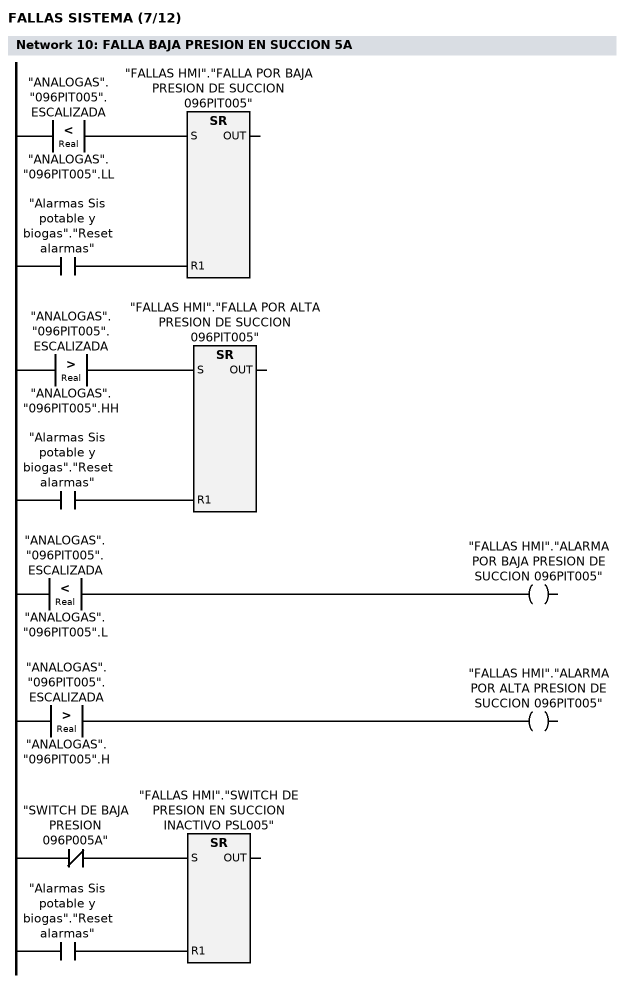
   RUNG wire#powerrail
      { S7_Templates := "SrcType := Real" } LT_Contact(in1 := "ANALOGAS"."096PIT005".ESCALIZADA, in2 := "ANALOGAS"."096PIT005".LL)
      S_SR(operand := "FALLAS HMI"."FALLA POR BAJA PRESION DE SUCCION 096PIT005", r1 := wire#w1)
   END_RUNG
   RUNG wire#powerrail
      Contact( "Alarmas Sis potable y biogas"."Reset alarmas" )
   END_RUNG wire#w1
   RUNG wire#powerrail
      { S7_Templates := "SrcType := Real" } GT_Contact(in1 := "ANALOGAS"."096PIT005".ESCALIZADA, in2 := "ANALOGAS"."096PIT005".HH)
      S_SR(operand := "FALLAS HMI"."FALLA POR ALTA PRESION DE SUCCION 096PIT005", r1 := wire#w2)
   END_RUNG
   RUNG wire#powerrail
      Contact( "Alarmas Sis potable y biogas"."Reset alarmas" )
   END_RUNG wire#w2
   RUNG wire#powerrail
      { S7_Templates := "SrcType := Real" } LT_Contact(in1 := "ANALOGAS"."096PIT005".ESCALIZADA, in2 := "ANALOGAS"."096PIT005".L)
      Coil( "FALLAS HMI"."ALARMA POR BAJA PRESION DE SUCCION 096PIT005" )
   END_RUNG
   RUNG wire#powerrail
      { S7_Templates := "SrcType := Real" } GT_Contact(in1 := "ANALOGAS"."096PIT005".ESCALIZADA, in2 := "ANALOGAS"."096PIT005".H)
      Coil( "FALLAS HMI"."ALARMA POR ALTA PRESION DE SUCCION 096PIT005" )
   END_RUNG
   RUNG wire#powerrail
      I_Contact( "SWITCH DE BAJA PRESION 096P005A" )
      S_SR(operand := "FALLAS HMI"."SWITCH DE PRESION EN SUCCION INACTIVO PSL005", r1 := wire#w3)
   END_RUNG
   RUNG wire#powerrail
      Contact( "Alarmas Sis potable y biogas"."Reset alarmas" )
   END_RUNG wire#w3
   // the same network as SCL:
   IF "ANALOGAS"."096PIT005".ESCALIZADA < "ANALOGAS"."096PIT005".LL THEN
       "FALLAS HMI"."FALLA POR BAJA PRESION DE SUCCION 096PIT005" := TRUE;   // SR flip-flop
   END_IF;
   IF "Alarmas Sis potable y biogas"."Reset alarmas" THEN
       "FALLAS HMI"."FALLA POR BAJA PRESION DE SUCCION 096PIT005" := FALSE;
   END_IF;
   IF "ANALOGAS"."096PIT005".ESCALIZADA > "ANALOGAS"."096PIT005".HH THEN
       "FALLAS HMI"."FALLA POR ALTA PRESION DE SUCCION 096PIT005" := TRUE;   // SR flip-flop
   END_IF;
   IF "Alarmas Sis potable y biogas"."Reset alarmas" THEN
       "FALLAS HMI"."FALLA POR ALTA PRESION DE SUCCION 096PIT005" := FALSE;
   END_IF;
   "FALLAS HMI"."ALARMA POR BAJA PRESION DE SUCCION 096PIT005" := "ANALOGAS"."096PIT005".ESCALIZADA < "ANALOGAS"."096PIT005".L;
   "FALLAS HMI"."ALARMA POR ALTA PRESION DE SUCCION 096PIT005" := "ANALOGAS"."096PIT005".ESCALIZADA > "ANALOGAS"."096PIT005".H;
   IF NOT "SWITCH DE BAJA PRESION 096P005A" THEN
       "FALLAS HMI"."SWITCH DE PRESION EN SUCCION INACTIVO PSL005" := TRUE;   // SR flip-flop
   END_IF;
   IF "Alarmas Sis potable y biogas"."Reset alarmas" THEN
       "FALLAS HMI"."SWITCH DE PRESION EN SUCCION INACTIVO PSL005" := FALSE;
   END_IF;
END_REGION

REGION Network 11: FALLA BAJA PRESION EN SUCCION 5B
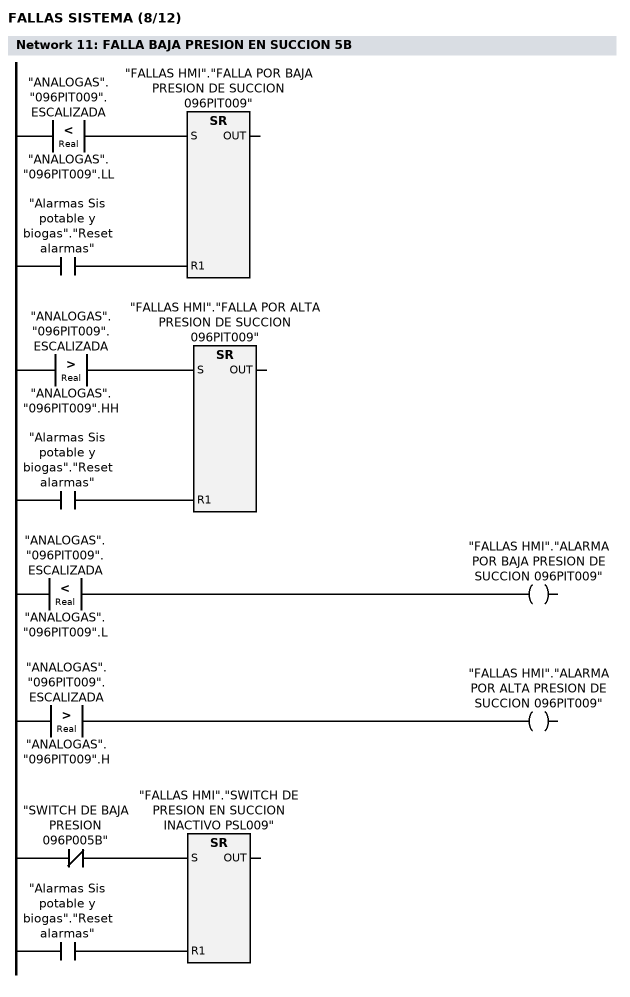
   RUNG wire#powerrail
      { S7_Templates := "SrcType := Real" } LT_Contact(in1 := "ANALOGAS"."096PIT009".ESCALIZADA, in2 := "ANALOGAS"."096PIT009".LL)
      S_SR(operand := "FALLAS HMI"."FALLA POR BAJA PRESION DE SUCCION 096PIT009", r1 := wire#w1)
   END_RUNG
   RUNG wire#powerrail
      Contact( "Alarmas Sis potable y biogas"."Reset alarmas" )
   END_RUNG wire#w1
   RUNG wire#powerrail
      { S7_Templates := "SrcType := Real" } GT_Contact(in1 := "ANALOGAS"."096PIT009".ESCALIZADA, in2 := "ANALOGAS"."096PIT009".HH)
      S_SR(operand := "FALLAS HMI"."FALLA POR ALTA PRESION DE SUCCION 096PIT009", r1 := wire#w2)
   END_RUNG
   RUNG wire#powerrail
      Contact( "Alarmas Sis potable y biogas"."Reset alarmas" )
   END_RUNG wire#w2
   RUNG wire#powerrail
      { S7_Templates := "SrcType := Real" } LT_Contact(in1 := "ANALOGAS"."096PIT009".ESCALIZADA, in2 := "ANALOGAS"."096PIT009".L)
      Coil( "FALLAS HMI"."ALARMA POR BAJA PRESION DE SUCCION 096PIT009" )
   END_RUNG
   RUNG wire#powerrail
      { S7_Templates := "SrcType := Real" } GT_Contact(in1 := "ANALOGAS"."096PIT009".ESCALIZADA, in2 := "ANALOGAS"."096PIT009".H)
      Coil( "FALLAS HMI"."ALARMA POR ALTA PRESION DE SUCCION 096PIT009" )
   END_RUNG
   RUNG wire#powerrail
      I_Contact( "SWITCH DE BAJA PRESION 096P005B" )
      S_SR(operand := "FALLAS HMI"."SWITCH DE PRESION EN SUCCION INACTIVO PSL009", r1 := wire#w3)
   END_RUNG
   RUNG wire#powerrail
      Contact( "Alarmas Sis potable y biogas"."Reset alarmas" )
   END_RUNG wire#w3
   // the same network as SCL:
   IF "ANALOGAS"."096PIT009".ESCALIZADA < "ANALOGAS"."096PIT009".LL THEN
       "FALLAS HMI"."FALLA POR BAJA PRESION DE SUCCION 096PIT009" := TRUE;   // SR flip-flop
   END_IF;
   IF "Alarmas Sis potable y biogas"."Reset alarmas" THEN
       "FALLAS HMI"."FALLA POR BAJA PRESION DE SUCCION 096PIT009" := FALSE;
   END_IF;
   IF "ANALOGAS"."096PIT009".ESCALIZADA > "ANALOGAS"."096PIT009".HH THEN
       "FALLAS HMI"."FALLA POR ALTA PRESION DE SUCCION 096PIT009" := TRUE;   // SR flip-flop
   END_IF;
   IF "Alarmas Sis potable y biogas"."Reset alarmas" THEN
       "FALLAS HMI"."FALLA POR ALTA PRESION DE SUCCION 096PIT009" := FALSE;
   END_IF;
   "FALLAS HMI"."ALARMA POR BAJA PRESION DE SUCCION 096PIT009" := "ANALOGAS"."096PIT009".ESCALIZADA < "ANALOGAS"."096PIT009".L;
   "FALLAS HMI"."ALARMA POR ALTA PRESION DE SUCCION 096PIT009" := "ANALOGAS"."096PIT009".ESCALIZADA > "ANALOGAS"."096PIT009".H;
   IF NOT "SWITCH DE BAJA PRESION 096P005B" THEN
       "FALLAS HMI"."SWITCH DE PRESION EN SUCCION INACTIVO PSL009" := TRUE;   // SR flip-flop
   END_IF;
   IF "Alarmas Sis potable y biogas"."Reset alarmas" THEN
       "FALLAS HMI"."SWITCH DE PRESION EN SUCCION INACTIVO PSL009" := FALSE;
   END_IF;
END_REGION

REGION Network 12: FALLA BAJA PRESION EN DESCARGA POTABLE
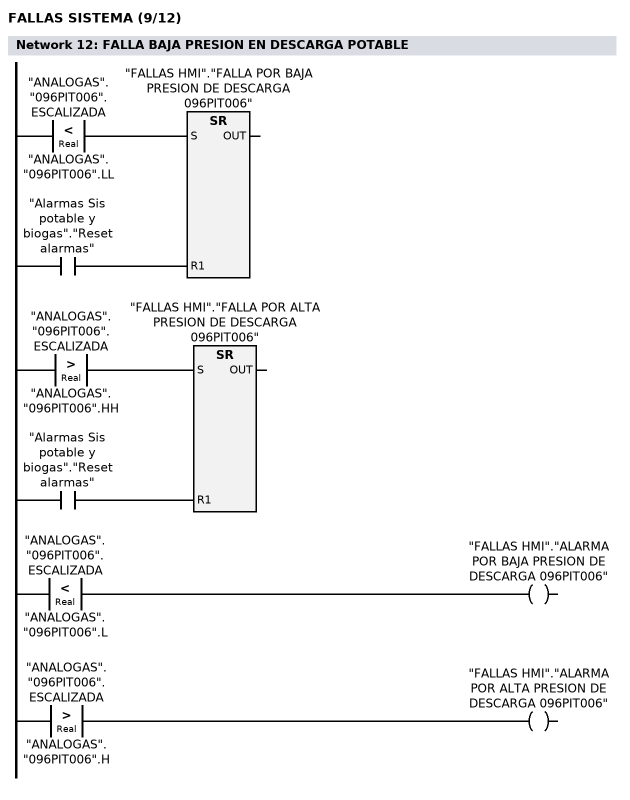
   RUNG wire#powerrail
      { S7_Templates := "SrcType := Real" } LT_Contact(in1 := "ANALOGAS"."096PIT006".ESCALIZADA, in2 := "ANALOGAS"."096PIT006".LL)
      S_SR(operand := "FALLAS HMI"."FALLA POR BAJA PRESION DE DESCARGA 096PIT006", r1 := wire#w1)
   END_RUNG
   RUNG wire#powerrail
      Contact( "Alarmas Sis potable y biogas"."Reset alarmas" )
   END_RUNG wire#w1
   RUNG wire#powerrail
      { S7_Templates := "SrcType := Real" } GT_Contact(in1 := "ANALOGAS"."096PIT006".ESCALIZADA, in2 := "ANALOGAS"."096PIT006".HH)
      S_SR(operand := "FALLAS HMI"."FALLA POR ALTA PRESION DE DESCARGA 096PIT006", r1 := wire#w2)
   END_RUNG
   RUNG wire#powerrail
      Contact( "Alarmas Sis potable y biogas"."Reset alarmas" )
   END_RUNG wire#w2
   RUNG wire#powerrail
      { S7_Templates := "SrcType := Real" } LT_Contact(in1 := "ANALOGAS"."096PIT006".ESCALIZADA, in2 := "ANALOGAS"."096PIT006".L)
      Coil( "FALLAS HMI"."ALARMA POR BAJA PRESION DE DESCARGA 096PIT006" )
   END_RUNG
   RUNG wire#powerrail
      { S7_Templates := "SrcType := Real" } GT_Contact(in1 := "ANALOGAS"."096PIT006".ESCALIZADA, in2 := "ANALOGAS"."096PIT006".H)
      Coil( "FALLAS HMI"."ALARMA POR ALTA PRESION DE DESCARGA 096PIT006" )
   END_RUNG
   // the same network as SCL:
   IF "ANALOGAS"."096PIT006".ESCALIZADA < "ANALOGAS"."096PIT006".LL THEN
       "FALLAS HMI"."FALLA POR BAJA PRESION DE DESCARGA 096PIT006" := TRUE;   // SR flip-flop
   END_IF;
   IF "Alarmas Sis potable y biogas"."Reset alarmas" THEN
       "FALLAS HMI"."FALLA POR BAJA PRESION DE DESCARGA 096PIT006" := FALSE;
   END_IF;
   IF "ANALOGAS"."096PIT006".ESCALIZADA > "ANALOGAS"."096PIT006".HH THEN
       "FALLAS HMI"."FALLA POR ALTA PRESION DE DESCARGA 096PIT006" := TRUE;   // SR flip-flop
   END_IF;
   IF "Alarmas Sis potable y biogas"."Reset alarmas" THEN
       "FALLAS HMI"."FALLA POR ALTA PRESION DE DESCARGA 096PIT006" := FALSE;
   END_IF;
   "FALLAS HMI"."ALARMA POR BAJA PRESION DE DESCARGA 096PIT006" := "ANALOGAS"."096PIT006".ESCALIZADA < "ANALOGAS"."096PIT006".L;
   "FALLAS HMI"."ALARMA POR ALTA PRESION DE DESCARGA 096PIT006" := "ANALOGAS"."096PIT006".ESCALIZADA > "ANALOGAS"."096PIT006".H;
END_REGION

REGION Network 13: FALLA BAJA PRESION EN DESCARGA 5A
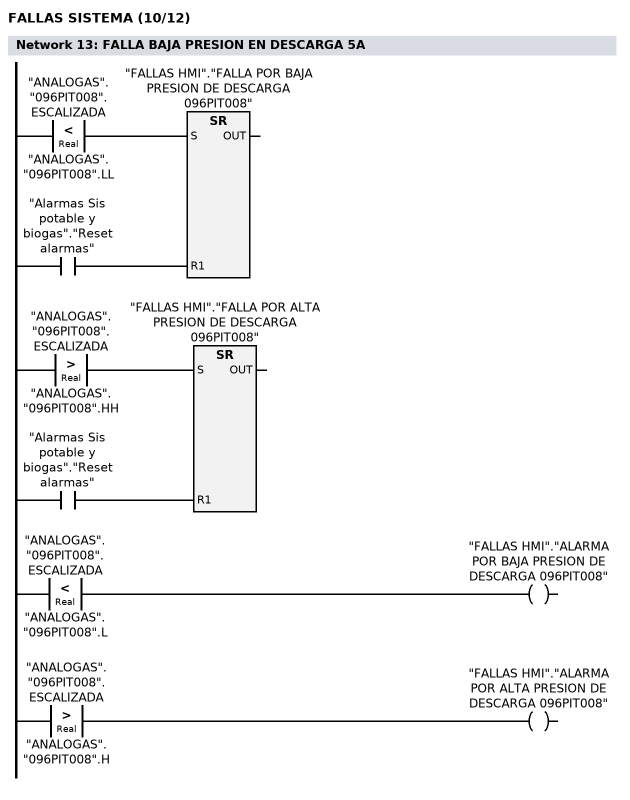
   RUNG wire#powerrail
      { S7_Templates := "SrcType := Real" } LT_Contact(in1 := "ANALOGAS"."096PIT008".ESCALIZADA, in2 := "ANALOGAS"."096PIT008".LL)
      S_SR(operand := "FALLAS HMI"."FALLA POR BAJA PRESION DE DESCARGA 096PIT008", r1 := wire#w1)
   END_RUNG
   RUNG wire#powerrail
      Contact( "Alarmas Sis potable y biogas"."Reset alarmas" )
   END_RUNG wire#w1
   RUNG wire#powerrail
      { S7_Templates := "SrcType := Real" } GT_Contact(in1 := "ANALOGAS"."096PIT008".ESCALIZADA, in2 := "ANALOGAS"."096PIT008".HH)
      S_SR(operand := "FALLAS HMI"."FALLA POR ALTA PRESION DE DESCARGA 096PIT008", r1 := wire#w2)
   END_RUNG
   RUNG wire#powerrail
      Contact( "Alarmas Sis potable y biogas"."Reset alarmas" )
   END_RUNG wire#w2
   RUNG wire#powerrail
      { S7_Templates := "SrcType := Real" } LT_Contact(in1 := "ANALOGAS"."096PIT008".ESCALIZADA, in2 := "ANALOGAS"."096PIT008".L)
      Coil( "FALLAS HMI"."ALARMA POR BAJA PRESION DE DESCARGA 096PIT008" )
   END_RUNG
   RUNG wire#powerrail
      { S7_Templates := "SrcType := Real" } GT_Contact(in1 := "ANALOGAS"."096PIT008".ESCALIZADA, in2 := "ANALOGAS"."096PIT008".H)
      Coil( "FALLAS HMI"."ALARMA POR ALTA PRESION DE DESCARGA 096PIT008" )
   END_RUNG
   // the same network as SCL:
   IF "ANALOGAS"."096PIT008".ESCALIZADA < "ANALOGAS"."096PIT008".LL THEN
       "FALLAS HMI"."FALLA POR BAJA PRESION DE DESCARGA 096PIT008" := TRUE;   // SR flip-flop
   END_IF;
   IF "Alarmas Sis potable y biogas"."Reset alarmas" THEN
       "FALLAS HMI"."FALLA POR BAJA PRESION DE DESCARGA 096PIT008" := FALSE;
   END_IF;
   IF "ANALOGAS"."096PIT008".ESCALIZADA > "ANALOGAS"."096PIT008".HH THEN
       "FALLAS HMI"."FALLA POR ALTA PRESION DE DESCARGA 096PIT008" := TRUE;   // SR flip-flop
   END_IF;
   IF "Alarmas Sis potable y biogas"."Reset alarmas" THEN
       "FALLAS HMI"."FALLA POR ALTA PRESION DE DESCARGA 096PIT008" := FALSE;
   END_IF;
   "FALLAS HMI"."ALARMA POR BAJA PRESION DE DESCARGA 096PIT008" := "ANALOGAS"."096PIT008".ESCALIZADA < "ANALOGAS"."096PIT008".L;
   "FALLAS HMI"."ALARMA POR ALTA PRESION DE DESCARGA 096PIT008" := "ANALOGAS"."096PIT008".ESCALIZADA > "ANALOGAS"."096PIT008".H;
END_REGION

REGION Network 14: FALLA BAJA PRESION EN DESCARGA 5B
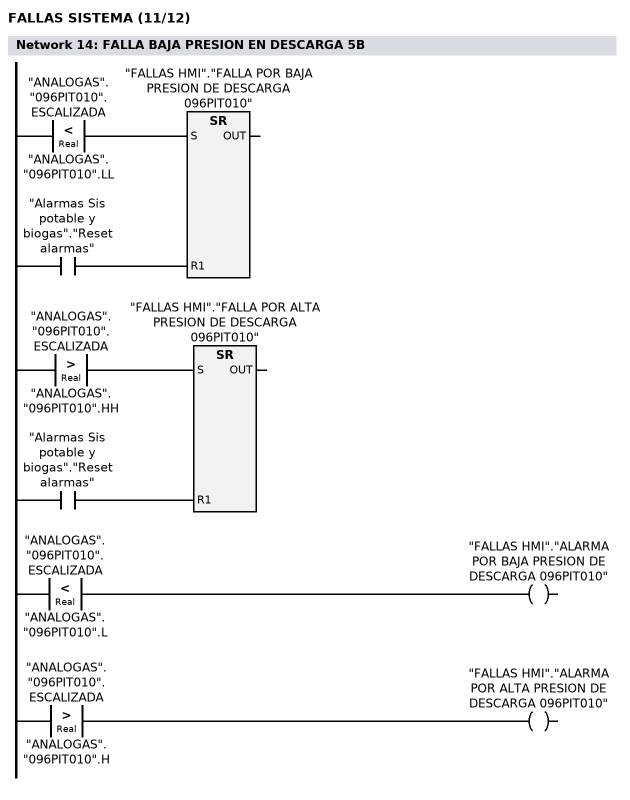
   RUNG wire#powerrail
      { S7_Templates := "SrcType := Real" } LT_Contact(in1 := "ANALOGAS"."096PIT010".ESCALIZADA, in2 := "ANALOGAS"."096PIT010".LL)
      S_SR(operand := "FALLAS HMI"."FALLA POR BAJA PRESION DE DESCARGA 096PIT010", r1 := wire#w1)
   END_RUNG
   RUNG wire#powerrail
      Contact( "Alarmas Sis potable y biogas"."Reset alarmas" )
   END_RUNG wire#w1
   RUNG wire#powerrail
      { S7_Templates := "SrcType := Real" } GT_Contact(in1 := "ANALOGAS"."096PIT010".ESCALIZADA, in2 := "ANALOGAS"."096PIT010".HH)
      S_SR(operand := "FALLAS HMI"."FALLA POR ALTA PRESION DE DESCARGA 096PIT010", r1 := wire#w2)
   END_RUNG
   RUNG wire#powerrail
      Contact( "Alarmas Sis potable y biogas"."Reset alarmas" )
   END_RUNG wire#w2
   RUNG wire#powerrail
      { S7_Templates := "SrcType := Real" } LT_Contact(in1 := "ANALOGAS"."096PIT010".ESCALIZADA, in2 := "ANALOGAS"."096PIT010".L)
      Coil( "FALLAS HMI"."ALARMA POR BAJA PRESION DE DESCARGA 096PIT010" )
   END_RUNG
   RUNG wire#powerrail
      { S7_Templates := "SrcType := Real" } GT_Contact(in1 := "ANALOGAS"."096PIT010".ESCALIZADA, in2 := "ANALOGAS"."096PIT010".H)
      Coil( "FALLAS HMI"."ALARMA POR ALTA PRESION DE DESCARGA 096PIT010" )
   END_RUNG
   // the same network as SCL:
   IF "ANALOGAS"."096PIT010".ESCALIZADA < "ANALOGAS"."096PIT010".LL THEN
       "FALLAS HMI"."FALLA POR BAJA PRESION DE DESCARGA 096PIT010" := TRUE;   // SR flip-flop
   END_IF;
   IF "Alarmas Sis potable y biogas"."Reset alarmas" THEN
       "FALLAS HMI"."FALLA POR BAJA PRESION DE DESCARGA 096PIT010" := FALSE;
   END_IF;
   IF "ANALOGAS"."096PIT010".ESCALIZADA > "ANALOGAS"."096PIT010".HH THEN
       "FALLAS HMI"."FALLA POR ALTA PRESION DE DESCARGA 096PIT010" := TRUE;   // SR flip-flop
   END_IF;
   IF "Alarmas Sis potable y biogas"."Reset alarmas" THEN
       "FALLAS HMI"."FALLA POR ALTA PRESION DE DESCARGA 096PIT010" := FALSE;
   END_IF;
   "FALLAS HMI"."ALARMA POR BAJA PRESION DE DESCARGA 096PIT010" := "ANALOGAS"."096PIT010".ESCALIZADA < "ANALOGAS"."096PIT010".L;
   "FALLAS HMI"."ALARMA POR ALTA PRESION DE DESCARGA 096PIT010" := "ANALOGAS"."096PIT010".ESCALIZADA > "ANALOGAS"."096PIT010".H;
END_REGION

REGION Network 15: FALLAS GRAL
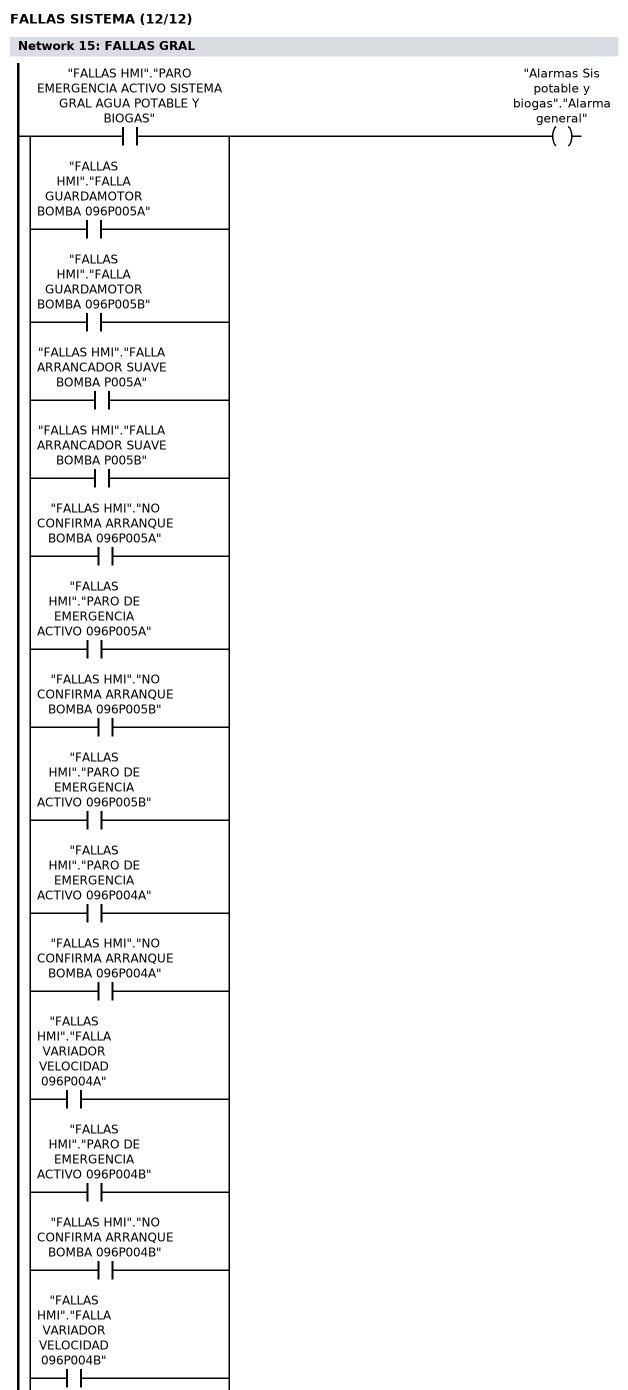
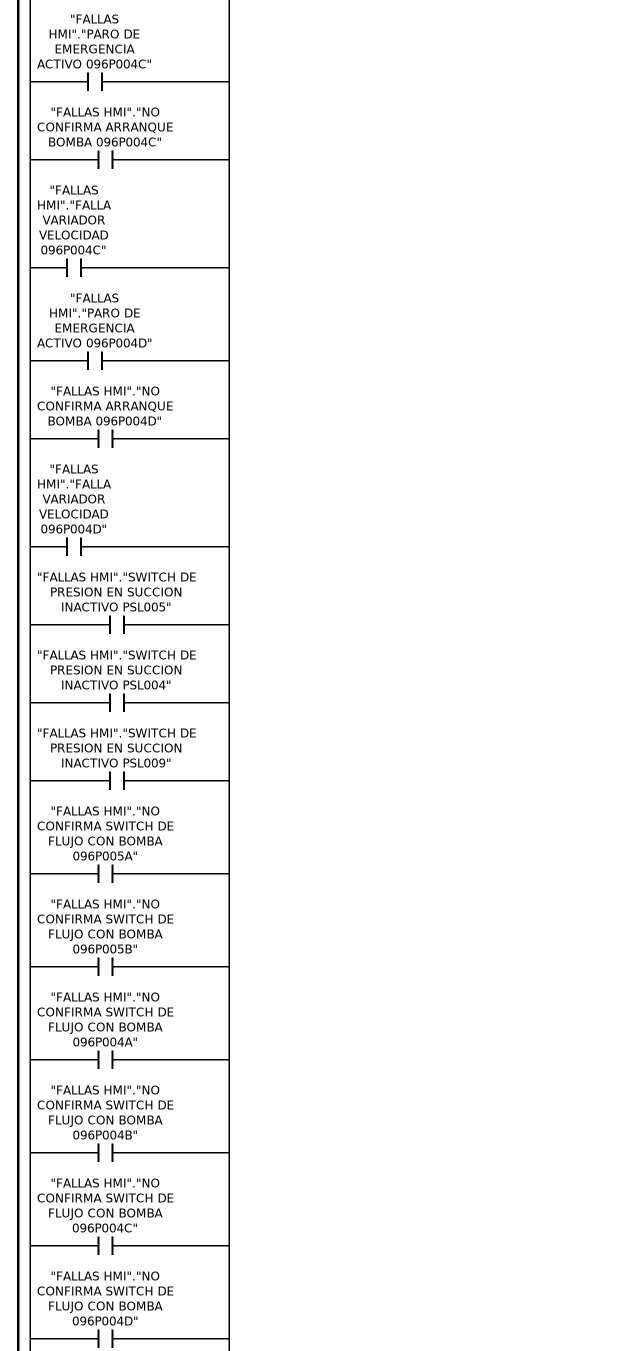
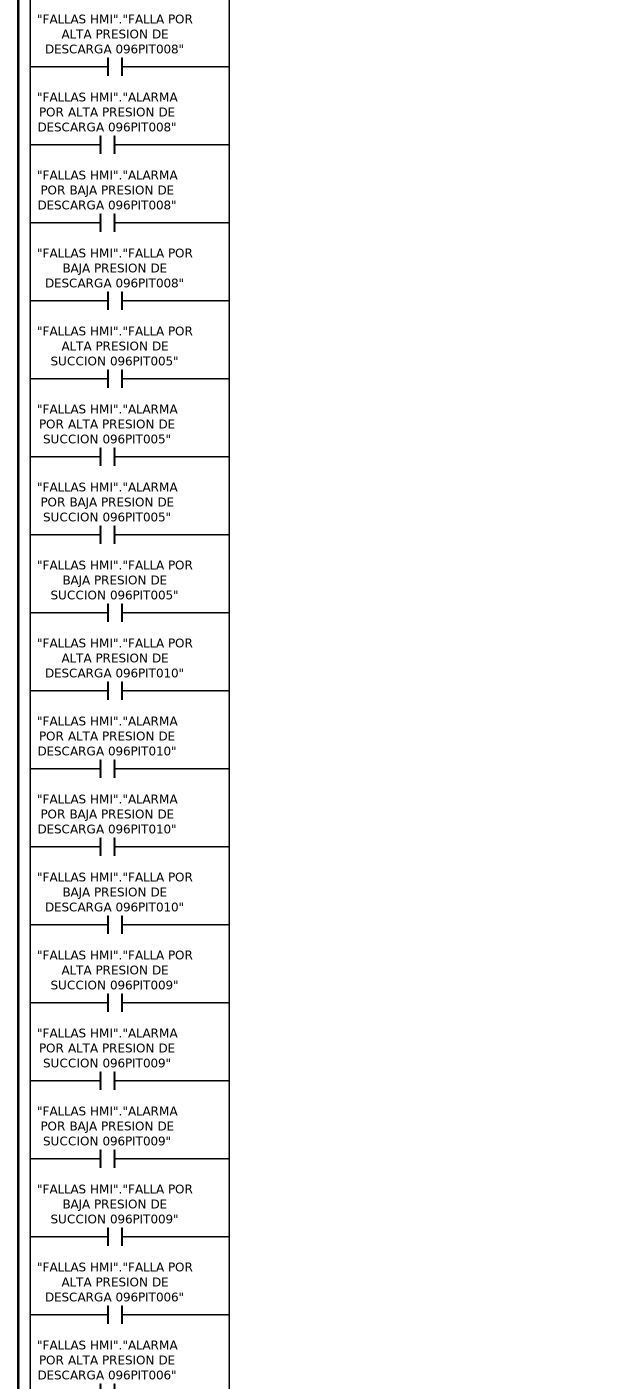
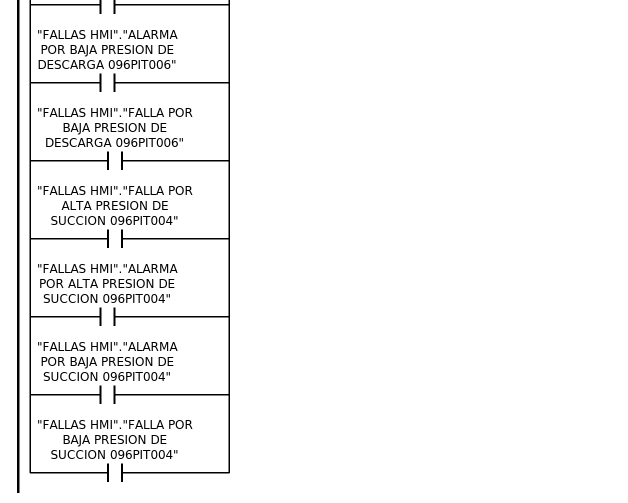
   RUNG wire#powerrail
      Contact( "FALLAS HMI"."PARO EMERGENCIA ACTIVO SISTEMA GRAL AGUA POTABLE Y BIOGAS" )
      wire#w1
      Coil( "Alarmas Sis potable y biogas"."Alarma general" )
   END_RUNG
   RUNG wire#powerrail
      Contact( "FALLAS HMI"."FALLA GUARDAMOTOR BOMBA 096P005A" )
   END_RUNG wire#w1
   RUNG wire#powerrail
      Contact( "FALLAS HMI"."FALLA GUARDAMOTOR BOMBA 096P005B" )
   END_RUNG wire#w1
   RUNG wire#powerrail
      Contact( "FALLAS HMI"."FALLA ARRANCADOR SUAVE BOMBA P005A" )
   END_RUNG wire#w1
   RUNG wire#powerrail
      Contact( "FALLAS HMI"."FALLA ARRANCADOR SUAVE BOMBA P005B" )
   END_RUNG wire#w1
   RUNG wire#powerrail
      Contact( "FALLAS HMI"."NO CONFIRMA ARRANQUE BOMBA 096P005A" )
   END_RUNG wire#w1
   RUNG wire#powerrail
      Contact( "FALLAS HMI"."PARO DE EMERGENCIA ACTIVO 096P005A" )
   END_RUNG wire#w1
   RUNG wire#powerrail
      Contact( "FALLAS HMI"."NO CONFIRMA ARRANQUE BOMBA 096P005B" )
   END_RUNG wire#w1
   RUNG wire#powerrail
      Contact( "FALLAS HMI"."PARO DE EMERGENCIA ACTIVO 096P005B" )
   END_RUNG wire#w1
   RUNG wire#powerrail
      Contact( "FALLAS HMI"."PARO DE EMERGENCIA ACTIVO 096P004A" )
   END_RUNG wire#w1
   RUNG wire#powerrail
      Contact( "FALLAS HMI"."NO CONFIRMA ARRANQUE BOMBA 096P004A" )
   END_RUNG wire#w1
   RUNG wire#powerrail
      Contact( "FALLAS HMI"."FALLA VARIADOR VELOCIDAD 096P004A" )
   END_RUNG wire#w1
   RUNG wire#powerrail
      Contact( "FALLAS HMI"."PARO DE EMERGENCIA ACTIVO 096P004B" )
   END_RUNG wire#w1
   RUNG wire#powerrail
      Contact( "FALLAS HMI"."NO CONFIRMA ARRANQUE BOMBA 096P004B" )
   END_RUNG wire#w1
   RUNG wire#powerrail
      Contact( "FALLAS HMI"."FALLA VARIADOR VELOCIDAD 096P004B" )
   END_RUNG wire#w1
   RUNG wire#powerrail
      Contact( "FALLAS HMI"."PARO DE EMERGENCIA ACTIVO 096P004C" )
   END_RUNG wire#w1
   RUNG wire#powerrail
      Contact( "FALLAS HMI"."NO CONFIRMA ARRANQUE BOMBA 096P004C" )
   END_RUNG wire#w1
   RUNG wire#powerrail
      Contact( "FALLAS HMI"."FALLA VARIADOR VELOCIDAD 096P004C" )
   END_RUNG wire#w1
   RUNG wire#powerrail
      Contact( "FALLAS HMI"."PARO DE EMERGENCIA ACTIVO 096P004D" )
   END_RUNG wire#w1
   RUNG wire#powerrail
      Contact( "FALLAS HMI"."NO CONFIRMA ARRANQUE BOMBA 096P004D" )
   END_RUNG wire#w1
   RUNG wire#powerrail
      Contact( "FALLAS HMI"."FALLA VARIADOR VELOCIDAD 096P004D" )
   END_RUNG wire#w1
   RUNG wire#powerrail
      Contact( "FALLAS HMI"."SWITCH DE PRESION EN SUCCION INACTIVO PSL005" )
   END_RUNG wire#w1
   RUNG wire#powerrail
      Contact( "FALLAS HMI"."SWITCH DE PRESION EN SUCCION INACTIVO PSL004" )
   END_RUNG wire#w1
   RUNG wire#powerrail
      Contact( "FALLAS HMI"."SWITCH DE PRESION EN SUCCION INACTIVO PSL009" )
   END_RUNG wire#w1
   RUNG wire#powerrail
      Contact( "FALLAS HMI"."NO CONFIRMA SWITCH DE FLUJO CON BOMBA 096P005A" )
   END_RUNG wire#w1
   RUNG wire#powerrail
      Contact( "FALLAS HMI"."NO CONFIRMA SWITCH DE FLUJO CON BOMBA 096P005B" )
   END_RUNG wire#w1
   RUNG wire#powerrail
      Contact( "FALLAS HMI"."NO CONFIRMA SWITCH DE FLUJO CON BOMBA 096P004A" )
   END_RUNG wire#w1
   RUNG wire#powerrail
      Contact( "FALLAS HMI"."NO CONFIRMA SWITCH DE FLUJO CON BOMBA 096P004B" )
   END_RUNG wire#w1
   RUNG wire#powerrail
      Contact( "FALLAS HMI"."NO CONFIRMA SWITCH DE FLUJO CON BOMBA 096P004C" )
   END_RUNG wire#w1
   RUNG wire#powerrail
      Contact( "FALLAS HMI"."NO CONFIRMA SWITCH DE FLUJO CON BOMBA 096P004D" )
   END_RUNG wire#w1
   RUNG wire#powerrail
      Contact( "FALLAS HMI"."FALLA POR ALTA PRESION DE DESCARGA 096PIT008" )
   END_RUNG wire#w1
   RUNG wire#powerrail
      Contact( "FALLAS HMI"."ALARMA POR ALTA PRESION DE DESCARGA 096PIT008" )
   END_RUNG wire#w1
   RUNG wire#powerrail
      Contact( "FALLAS HMI"."ALARMA POR BAJA PRESION DE DESCARGA 096PIT008" )
   END_RUNG wire#w1
   RUNG wire#powerrail
      Contact( "FALLAS HMI"."FALLA POR BAJA PRESION DE DESCARGA 096PIT008" )
   END_RUNG wire#w1
   RUNG wire#powerrail
      Contact( "FALLAS HMI"."FALLA POR ALTA PRESION DE SUCCION 096PIT005" )
   END_RUNG wire#w1
   RUNG wire#powerrail
      Contact( "FALLAS HMI"."ALARMA POR ALTA PRESION DE SUCCION 096PIT005" )
   END_RUNG wire#w1
   RUNG wire#powerrail
      Contact( "FALLAS HMI"."ALARMA POR BAJA PRESION DE SUCCION 096PIT005" )
   END_RUNG wire#w1
   RUNG wire#powerrail
      Contact( "FALLAS HMI"."FALLA POR BAJA PRESION DE SUCCION 096PIT005" )
   END_RUNG wire#w1
   RUNG wire#powerrail
      Contact( "FALLAS HMI"."FALLA POR ALTA PRESION DE DESCARGA 096PIT010" )
   END_RUNG wire#w1
   RUNG wire#powerrail
      Contact( "FALLAS HMI"."ALARMA POR ALTA PRESION DE DESCARGA 096PIT010" )
   END_RUNG wire#w1
   RUNG wire#powerrail
      Contact( "FALLAS HMI"."ALARMA POR BAJA PRESION DE DESCARGA 096PIT010" )
   END_RUNG wire#w1
   RUNG wire#powerrail
      Contact( "FALLAS HMI"."FALLA POR BAJA PRESION DE DESCARGA 096PIT010" )
   END_RUNG wire#w1
   RUNG wire#powerrail
      Contact( "FALLAS HMI"."FALLA POR ALTA PRESION DE SUCCION 096PIT009" )
   END_RUNG wire#w1
   RUNG wire#powerrail
      Contact( "FALLAS HMI"."ALARMA POR ALTA PRESION DE SUCCION 096PIT009" )
   END_RUNG wire#w1
   RUNG wire#powerrail
      Contact( "FALLAS HMI"."ALARMA POR BAJA PRESION DE SUCCION 096PIT009" )
   END_RUNG wire#w1
   RUNG wire#powerrail
      Contact( "FALLAS HMI"."FALLA POR BAJA PRESION DE SUCCION 096PIT009" )
   END_RUNG wire#w1
   RUNG wire#powerrail
      Contact( "FALLAS HMI"."FALLA POR ALTA PRESION DE DESCARGA 096PIT006" )
   END_RUNG wire#w1
   RUNG wire#powerrail
      Contact( "FALLAS HMI"."ALARMA POR ALTA PRESION DE DESCARGA 096PIT006" )
   END_RUNG wire#w1
   RUNG wire#powerrail
      Contact( "FALLAS HMI"."ALARMA POR BAJA PRESION DE DESCARGA 096PIT006" )
   END_RUNG wire#w1
   RUNG wire#powerrail
      Contact( "FALLAS HMI"."FALLA POR BAJA PRESION DE DESCARGA 096PIT006" )
   END_RUNG wire#w1
   RUNG wire#powerrail
      Contact( "FALLAS HMI"."FALLA POR ALTA PRESION DE SUCCION 096PIT004" )
   END_RUNG wire#w1
   RUNG wire#powerrail
      Contact( "FALLAS HMI"."ALARMA POR ALTA PRESION DE SUCCION 096PIT004" )
   END_RUNG wire#w1
   RUNG wire#powerrail
      Contact( "FALLAS HMI"."ALARMA POR BAJA PRESION DE SUCCION 096PIT004" )
   END_RUNG wire#w1
   RUNG wire#powerrail
      Contact( "FALLAS HMI"."FALLA POR BAJA PRESION DE SUCCION 096PIT004" )
   END_RUNG wire#w1
   // the same network as SCL:
   "Alarmas Sis potable y biogas"."Alarma general" := "FALLAS HMI"."PARO EMERGENCIA ACTIVO SISTEMA GRAL AGUA POTABLE Y BIOGAS" OR "FALLAS HMI"."FALLA GUARDAMOTOR BOMBA 096P005A" OR "FALLAS HMI"."FALLA GUARDAMOTOR BOMBA 096P005B" OR "FALLAS HMI"."FALLA ARRANCADOR SUAVE BOMBA P005A" OR "FALLAS HMI"."FALLA ARRANCADOR SUAVE BOMBA P005B" OR "FALLAS HMI"."NO CONFIRMA ARRANQUE BOMBA 096P005A" OR "FALLAS HMI"."PARO DE EMERGENCIA ACTIVO 096P005A" OR "FALLAS HMI"."NO CONFIRMA ARRANQUE BOMBA 096P005B" OR "FALLAS HMI"."PARO DE EMERGENCIA ACTIVO 096P005B" OR "FALLAS HMI"."PARO DE EMERGENCIA ACTIVO 096P004A" OR "FALLAS HMI"."NO CONFIRMA ARRANQUE BOMBA 096P004A" OR "FALLAS HMI"."FALLA VARIADOR VELOCIDAD 096P004A" OR "FALLAS HMI"."PARO DE EMERGENCIA ACTIVO 096P004B" OR "FALLAS HMI"."NO CONFIRMA ARRANQUE BOMBA 096P004B" OR "FALLAS HMI"."FALLA VARIADOR VELOCIDAD 096P004B" OR "FALLAS HMI"."PARO DE EMERGENCIA ACTIVO 096P004C" OR "FALLAS HMI"."NO CONFIRMA ARRANQUE BOMBA 096P004C" OR "FALLAS HMI"."FALLA VARIADOR VELOCIDAD 096P004C" OR "FALLAS HMI"."PARO DE EMERGENCIA ACTIVO 096P004D" OR "FALLAS HMI"."NO CONFIRMA ARRANQUE BOMBA 096P004D" OR "FALLAS HMI"."FALLA VARIADOR VELOCIDAD 096P004D" OR "FALLAS HMI"."SWITCH DE PRESION EN SUCCION INACTIVO PSL005" OR "FALLAS HMI"."SWITCH DE PRESION EN SUCCION INACTIVO PSL004" OR "FALLAS HMI"."SWITCH DE PRESION EN SUCCION INACTIVO PSL009" OR "FALLAS HMI"."NO CONFIRMA SWITCH DE FLUJO CON BOMBA 096P005A" OR "FALLAS HMI"."NO CONFIRMA SWITCH DE FLUJO CON BOMBA 096P005B" OR "FALLAS HMI"."NO CONFIRMA SWITCH DE FLUJO CON BOMBA 096P004A" OR "FALLAS HMI"."NO CONFIRMA SWITCH DE FLUJO CON BOMBA 096P004B" OR "FALLAS HMI"."NO CONFIRMA SWITCH DE FLUJO CON BOMBA 096P004C" OR "FALLAS HMI"."NO CONFIRMA SWITCH DE FLUJO CON BOMBA 096P004D" OR "FALLAS HMI"."FALLA POR ALTA PRESION DE DESCARGA 096PIT008" OR "FALLAS HMI"."ALARMA POR ALTA PRESION DE DESCARGA 096PIT008" OR "FALLAS HMI"."ALARMA POR BAJA PRESION DE DESCARGA 096PIT008" OR "FALLAS HMI"."FALLA POR BAJA PRESION DE DESCARGA 096PIT008" OR "FALLAS HMI"."FALLA POR ALTA PRESION DE SUCCION 096PIT005" OR "FALLAS HMI"."ALARMA POR ALTA PRESION DE SUCCION 096PIT005" OR "FALLAS HMI"."ALARMA POR BAJA PRESION DE SUCCION 096PIT005" OR "FALLAS HMI"."FALLA POR BAJA PRESION DE SUCCION 096PIT005" OR "FALLAS HMI"."FALLA POR ALTA PRESION DE DESCARGA 096PIT010" OR "FALLAS HMI"."ALARMA POR ALTA PRESION DE DESCARGA 096PIT010" OR "FALLAS HMI"."ALARMA POR BAJA PRESION DE DESCARGA 096PIT010" OR "FALLAS HMI"."FALLA POR BAJA PRESION DE DESCARGA 096PIT010" OR "FALLAS HMI"."FALLA POR ALTA PRESION DE SUCCION 096PIT009" OR "FALLAS HMI"."ALARMA POR ALTA PRESION DE SUCCION 096PIT009" OR "FALLAS HMI"."ALARMA POR BAJA PRESION DE SUCCION 096PIT009" OR "FALLAS HMI"."FALLA POR BAJA PRESION DE SUCCION 096PIT009" OR "FALLAS HMI"."FALLA POR ALTA PRESION DE DESCARGA 096PIT006" OR "FALLAS HMI"."ALARMA POR ALTA PRESION DE DESCARGA 096PIT006" OR "FALLAS HMI"."ALARMA POR BAJA PRESION DE DESCARGA 096PIT006" OR "FALLAS HMI"."FALLA POR BAJA PRESION DE DESCARGA 096PIT006" OR "FALLAS HMI"."FALLA POR ALTA PRESION DE SUCCION 096PIT004" OR "FALLAS HMI"."ALARMA POR ALTA PRESION DE SUCCION 096PIT004" OR "FALLAS HMI"."ALARMA POR BAJA PRESION DE SUCCION 096PIT004" OR "FALLAS HMI"."FALLA POR BAJA PRESION DE SUCCION 096PIT004";
END_REGION
END_FUNCTION

FUNCTION "Esc Salidas Analogas" : Void   // FC12, LAD
{ S7_Optimized_Access := 'TRUE' }
VERSION : 0.1
   VAR_TEMP
      SA1 : Real;
      SA2 : Real;
      SA3 : Real;
      SA4 : Real;
      SA5 : Real;
      SA6 : Real;
      "CONSIGNA 1" : Real;
      "CONSIGNA 2" : Real;
      "CONSIGNA 3" : Real;
      "CONSIGNA 4" : Real;
      "CONSIGNA 5" : Real;
      "CONSIGNA 6" : Real;
   END_VAR
BEGIN

REGION Network 1: SALIDA ANALOGA 096P004A
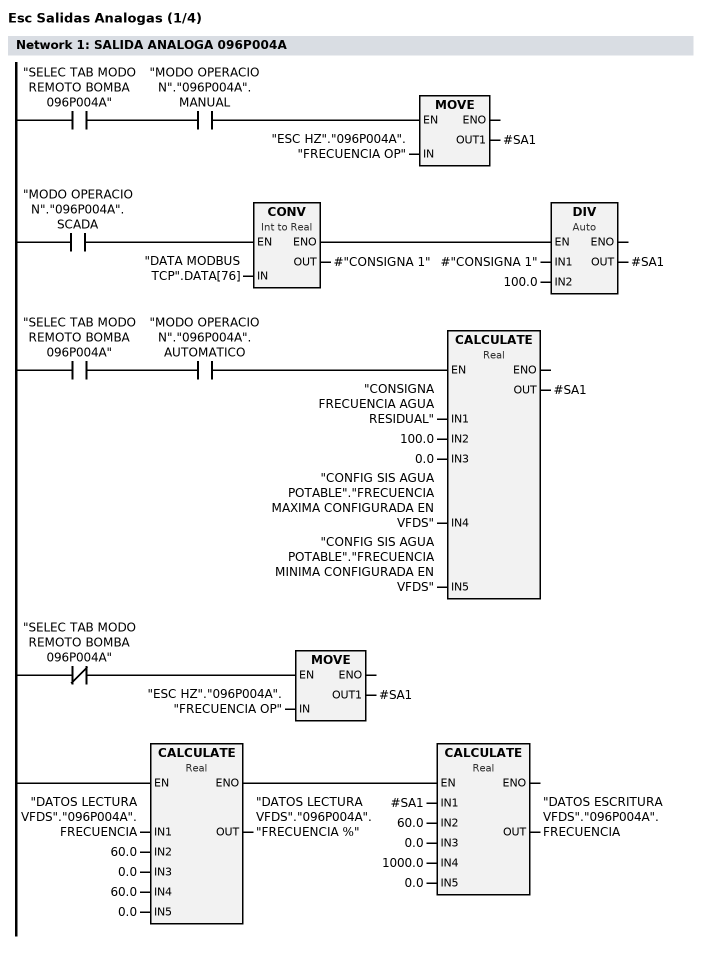
   RUNG wire#powerrail
      Contact( "SELEC TAB MODO REMOTO BOMBA 096P004A" )
      Contact( "MODO OPERACION"."096P004A".MANUAL )
      Move(in := "ESC HZ"."096P004A"."FRECUENCIA OP", out1 => #SA1)
   END_RUNG
   RUNG wire#powerrail
      Contact( "MODO OPERACION"."096P004A".SCADA )
      { S7_Templates := "[SrcType := Int, DestType := Real]" } Convert(in := "DATA MODBUS TCP".DATA[76], out => #"CONSIGNA 1")
      Div(in1 := #"CONSIGNA 1", in2 := 100.0, out => #SA1)
   END_RUNG
   RUNG wire#powerrail
      Contact( "SELEC TAB MODO REMOTO BOMBA 096P004A" )
      Contact( "MODO OPERACION"."096P004A".AUTOMATICO )
      { S7_Templates := "SrcType := Real"; S7_Expression := "(((IN4-IN5)/(IN2-IN3))*IN1)+(IN5-(((IN4-IN5)/(IN2-IN3))*IN3))" } Calculate(in1 := "CONSIGNA FRECUENCIA AGUA RESIDUAL", in2 := 100.0, in3 := 0.0, in4 := "CONFIG SIS AGUA POTABLE"."FRECUENCIA MAXIMA CONFIGURADA EN VFDS", in5 := "CONFIG SIS AGUA POTABLE"."FRECUENCIA MINIMA CONFIGURADA EN VFDS", out => #SA1)
   END_RUNG
   RUNG wire#powerrail
      I_Contact( "SELEC TAB MODO REMOTO BOMBA 096P004A" )
      Move(in := "ESC HZ"."096P004A"."FRECUENCIA OP", out1 => #SA1)
   END_RUNG
   RUNG wire#powerrail
      { S7_Templates := "SrcType := Real"; S7_Expression := "(((IN4-IN5)/(IN2-IN3))*IN1)+(IN5-(((IN4-IN5)/(IN2-IN3))*IN3))" } Calculate(in1 := "DATOS LECTURA VFDS"."096P004A".FRECUENCIA, in2 := 60.0, in3 := 0.0, in4 := 60.0, in5 := 0.0, out => "DATOS LECTURA VFDS"."096P004A"."FRECUENCIA %")
      { S7_Templates := "SrcType := Real"; S7_Expression := "(((IN4-IN5)/(IN2-IN3))*IN1)+(IN5-(((IN4-IN5)/(IN2-IN3))*IN3))" } Calculate(in1 := #SA1, in2 := 60.0, in3 := 0.0, in4 := 1000.0, in5 := 0.0, out => "DATOS ESCRITURA VFDS"."096P004A".FRECUENCIA)
   END_RUNG
   // the same network as SCL:
   IF "SELEC TAB MODO REMOTO BOMBA 096P004A" AND "MODO OPERACION"."096P004A".MANUAL THEN
       #SA1 := "ESC HZ"."096P004A"."FRECUENCIA OP";
   END_IF;
   IF "MODO OPERACION"."096P004A".SCADA THEN
       #"CONSIGNA 1" := INT_TO_REAL("DATA MODBUS TCP".DATA[76]);
       #SA1 := #"CONSIGNA 1" / 100.0;
   END_IF;
   IF "SELEC TAB MODO REMOTO BOMBA 096P004A" AND "MODO OPERACION"."096P004A".AUTOMATICO THEN
       #SA1 := ((("CONFIG SIS AGUA POTABLE"."FRECUENCIA MAXIMA CONFIGURADA EN VFDS"-"CONFIG SIS AGUA POTABLE"."FRECUENCIA MINIMA CONFIGURADA EN VFDS")/(100.0-0.0))*"CONSIGNA FRECUENCIA AGUA RESIDUAL")+("CONFIG SIS AGUA POTABLE"."FRECUENCIA MINIMA CONFIGURADA EN VFDS"-((("CONFIG SIS AGUA POTABLE"."FRECUENCIA MAXIMA CONFIGURADA EN VFDS"-"CONFIG SIS AGUA POTABLE"."FRECUENCIA MINIMA CONFIGURADA EN VFDS")/(100.0-0.0))*0.0));
   END_IF;
   IF NOT "SELEC TAB MODO REMOTO BOMBA 096P004A" THEN #SA1 := "ESC HZ"."096P004A"."FRECUENCIA OP"; END_IF;
   "DATOS LECTURA VFDS"."096P004A"."FRECUENCIA %" := (((60.0-0.0)/(60.0-0.0))*"DATOS LECTURA VFDS"."096P004A".FRECUENCIA)+(0.0-(((60.0-0.0)/(60.0-0.0))*0.0));
   "DATOS ESCRITURA VFDS"."096P004A".FRECUENCIA := (((1000.0-0.0)/(60.0-0.0))*#SA1)+(0.0-(((1000.0-0.0)/(60.0-0.0))*0.0));
END_REGION

REGION Network 2: SALIDA ANALOGA 096P004B
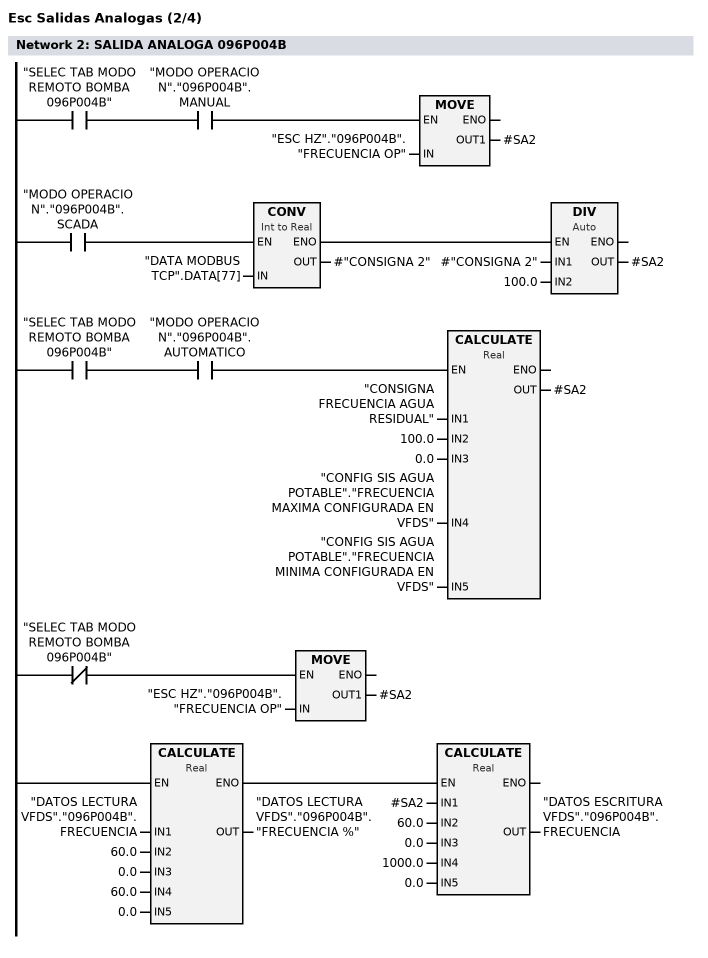
   RUNG wire#powerrail
      Contact( "SELEC TAB MODO REMOTO BOMBA 096P004B" )
      Contact( "MODO OPERACION"."096P004B".MANUAL )
      Move(in := "ESC HZ"."096P004B"."FRECUENCIA OP", out1 => #SA2)
   END_RUNG
   RUNG wire#powerrail
      Contact( "MODO OPERACION"."096P004B".SCADA )
      { S7_Templates := "[SrcType := Int, DestType := Real]" } Convert(in := "DATA MODBUS TCP".DATA[77], out => #"CONSIGNA 2")
      Div(in1 := #"CONSIGNA 2", in2 := 100.0, out => #SA2)
   END_RUNG
   RUNG wire#powerrail
      Contact( "SELEC TAB MODO REMOTO BOMBA 096P004B" )
      Contact( "MODO OPERACION"."096P004B".AUTOMATICO )
      { S7_Templates := "SrcType := Real"; S7_Expression := "(((IN4-IN5)/(IN2-IN3))*IN1)+(IN5-(((IN4-IN5)/(IN2-IN3))*IN3))" } Calculate(in1 := "CONSIGNA FRECUENCIA AGUA RESIDUAL", in2 := 100.0, in3 := 0.0, in4 := "CONFIG SIS AGUA POTABLE"."FRECUENCIA MAXIMA CONFIGURADA EN VFDS", in5 := "CONFIG SIS AGUA POTABLE"."FRECUENCIA MINIMA CONFIGURADA EN VFDS", out => #SA2)
   END_RUNG
   RUNG wire#powerrail
      I_Contact( "SELEC TAB MODO REMOTO BOMBA 096P004B" )
      Move(in := "ESC HZ"."096P004B"."FRECUENCIA OP", out1 => #SA2)
   END_RUNG
   RUNG wire#powerrail
      { S7_Templates := "SrcType := Real"; S7_Expression := "(((IN4-IN5)/(IN2-IN3))*IN1)+(IN5-(((IN4-IN5)/(IN2-IN3))*IN3))" } Calculate(in1 := "DATOS LECTURA VFDS"."096P004B".FRECUENCIA, in2 := 60.0, in3 := 0.0, in4 := 60.0, in5 := 0.0, out => "DATOS LECTURA VFDS"."096P004B"."FRECUENCIA %")
      { S7_Templates := "SrcType := Real"; S7_Expression := "(((IN4-IN5)/(IN2-IN3))*IN1)+(IN5-(((IN4-IN5)/(IN2-IN3))*IN3))" } Calculate(in1 := #SA2, in2 := 60.0, in3 := 0.0, in4 := 1000.0, in5 := 0.0, out => "DATOS ESCRITURA VFDS"."096P004B".FRECUENCIA)
   END_RUNG
   // the same network as SCL:
   IF "SELEC TAB MODO REMOTO BOMBA 096P004B" AND "MODO OPERACION"."096P004B".MANUAL THEN
       #SA2 := "ESC HZ"."096P004B"."FRECUENCIA OP";
   END_IF;
   IF "MODO OPERACION"."096P004B".SCADA THEN
       #"CONSIGNA 2" := INT_TO_REAL("DATA MODBUS TCP".DATA[77]);
       #SA2 := #"CONSIGNA 2" / 100.0;
   END_IF;
   IF "SELEC TAB MODO REMOTO BOMBA 096P004B" AND "MODO OPERACION"."096P004B".AUTOMATICO THEN
       #SA2 := ((("CONFIG SIS AGUA POTABLE"."FRECUENCIA MAXIMA CONFIGURADA EN VFDS"-"CONFIG SIS AGUA POTABLE"."FRECUENCIA MINIMA CONFIGURADA EN VFDS")/(100.0-0.0))*"CONSIGNA FRECUENCIA AGUA RESIDUAL")+("CONFIG SIS AGUA POTABLE"."FRECUENCIA MINIMA CONFIGURADA EN VFDS"-((("CONFIG SIS AGUA POTABLE"."FRECUENCIA MAXIMA CONFIGURADA EN VFDS"-"CONFIG SIS AGUA POTABLE"."FRECUENCIA MINIMA CONFIGURADA EN VFDS")/(100.0-0.0))*0.0));
   END_IF;
   IF NOT "SELEC TAB MODO REMOTO BOMBA 096P004B" THEN #SA2 := "ESC HZ"."096P004B"."FRECUENCIA OP"; END_IF;
   "DATOS LECTURA VFDS"."096P004B"."FRECUENCIA %" := (((60.0-0.0)/(60.0-0.0))*"DATOS LECTURA VFDS"."096P004B".FRECUENCIA)+(0.0-(((60.0-0.0)/(60.0-0.0))*0.0));
   "DATOS ESCRITURA VFDS"."096P004B".FRECUENCIA := (((1000.0-0.0)/(60.0-0.0))*#SA2)+(0.0-(((1000.0-0.0)/(60.0-0.0))*0.0));
END_REGION

REGION Network 3: SALIDA ANALOGA 096P004C
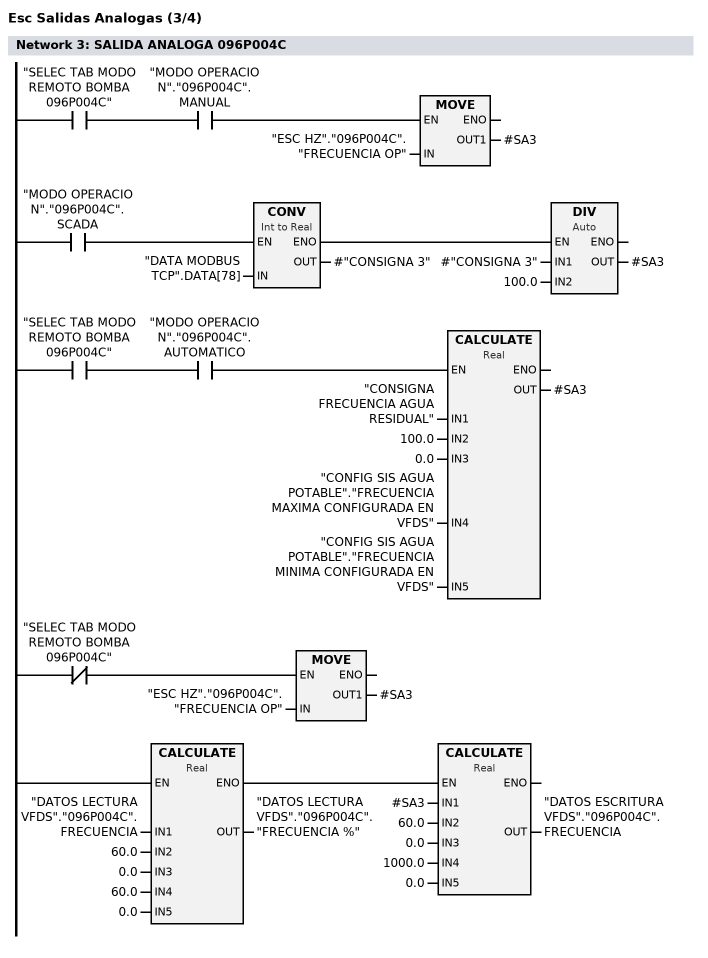
   RUNG wire#powerrail
      Contact( "SELEC TAB MODO REMOTO BOMBA 096P004C" )
      Contact( "MODO OPERACION"."096P004C".MANUAL )
      Move(in := "ESC HZ"."096P004C"."FRECUENCIA OP", out1 => #SA3)
   END_RUNG
   RUNG wire#powerrail
      Contact( "MODO OPERACION"."096P004C".SCADA )
      { S7_Templates := "[SrcType := Int, DestType := Real]" } Convert(in := "DATA MODBUS TCP".DATA[78], out => #"CONSIGNA 3")
      Div(in1 := #"CONSIGNA 3", in2 := 100.0, out => #SA3)
   END_RUNG
   RUNG wire#powerrail
      Contact( "SELEC TAB MODO REMOTO BOMBA 096P004C" )
      Contact( "MODO OPERACION"."096P004C".AUTOMATICO )
      { S7_Templates := "SrcType := Real"; S7_Expression := "(((IN4-IN5)/(IN2-IN3))*IN1)+(IN5-(((IN4-IN5)/(IN2-IN3))*IN3))" } Calculate(in1 := "CONSIGNA FRECUENCIA AGUA RESIDUAL", in2 := 100.0, in3 := 0.0, in4 := "CONFIG SIS AGUA POTABLE"."FRECUENCIA MAXIMA CONFIGURADA EN VFDS", in5 := "CONFIG SIS AGUA POTABLE"."FRECUENCIA MINIMA CONFIGURADA EN VFDS", out => #SA3)
   END_RUNG
   RUNG wire#powerrail
      I_Contact( "SELEC TAB MODO REMOTO BOMBA 096P004C" )
      Move(in := "ESC HZ"."096P004C"."FRECUENCIA OP", out1 => #SA3)
   END_RUNG
   RUNG wire#powerrail
      { S7_Templates := "SrcType := Real"; S7_Expression := "(((IN4-IN5)/(IN2-IN3))*IN1)+(IN5-(((IN4-IN5)/(IN2-IN3))*IN3))" } Calculate(in1 := "DATOS LECTURA VFDS"."096P004C".FRECUENCIA, in2 := 60.0, in3 := 0.0, in4 := 60.0, in5 := 0.0, out => "DATOS LECTURA VFDS"."096P004C"."FRECUENCIA %")
      { S7_Templates := "SrcType := Real"; S7_Expression := "(((IN4-IN5)/(IN2-IN3))*IN1)+(IN5-(((IN4-IN5)/(IN2-IN3))*IN3))" } Calculate(in1 := #SA3, in2 := 60.0, in3 := 0.0, in4 := 1000.0, in5 := 0.0, out => "DATOS ESCRITURA VFDS"."096P004C".FRECUENCIA)
   END_RUNG
   // the same network as SCL:
   IF "SELEC TAB MODO REMOTO BOMBA 096P004C" AND "MODO OPERACION"."096P004C".MANUAL THEN
       #SA3 := "ESC HZ"."096P004C"."FRECUENCIA OP";
   END_IF;
   IF "MODO OPERACION"."096P004C".SCADA THEN
       #"CONSIGNA 3" := INT_TO_REAL("DATA MODBUS TCP".DATA[78]);
       #SA3 := #"CONSIGNA 3" / 100.0;
   END_IF;
   IF "SELEC TAB MODO REMOTO BOMBA 096P004C" AND "MODO OPERACION"."096P004C".AUTOMATICO THEN
       #SA3 := ((("CONFIG SIS AGUA POTABLE"."FRECUENCIA MAXIMA CONFIGURADA EN VFDS"-"CONFIG SIS AGUA POTABLE"."FRECUENCIA MINIMA CONFIGURADA EN VFDS")/(100.0-0.0))*"CONSIGNA FRECUENCIA AGUA RESIDUAL")+("CONFIG SIS AGUA POTABLE"."FRECUENCIA MINIMA CONFIGURADA EN VFDS"-((("CONFIG SIS AGUA POTABLE"."FRECUENCIA MAXIMA CONFIGURADA EN VFDS"-"CONFIG SIS AGUA POTABLE"."FRECUENCIA MINIMA CONFIGURADA EN VFDS")/(100.0-0.0))*0.0));
   END_IF;
   IF NOT "SELEC TAB MODO REMOTO BOMBA 096P004C" THEN #SA3 := "ESC HZ"."096P004C"."FRECUENCIA OP"; END_IF;
   "DATOS LECTURA VFDS"."096P004C"."FRECUENCIA %" := (((60.0-0.0)/(60.0-0.0))*"DATOS LECTURA VFDS"."096P004C".FRECUENCIA)+(0.0-(((60.0-0.0)/(60.0-0.0))*0.0));
   "DATOS ESCRITURA VFDS"."096P004C".FRECUENCIA := (((1000.0-0.0)/(60.0-0.0))*#SA3)+(0.0-(((1000.0-0.0)/(60.0-0.0))*0.0));
END_REGION

REGION Network 4: SALIDA ANALOGA 096P004D
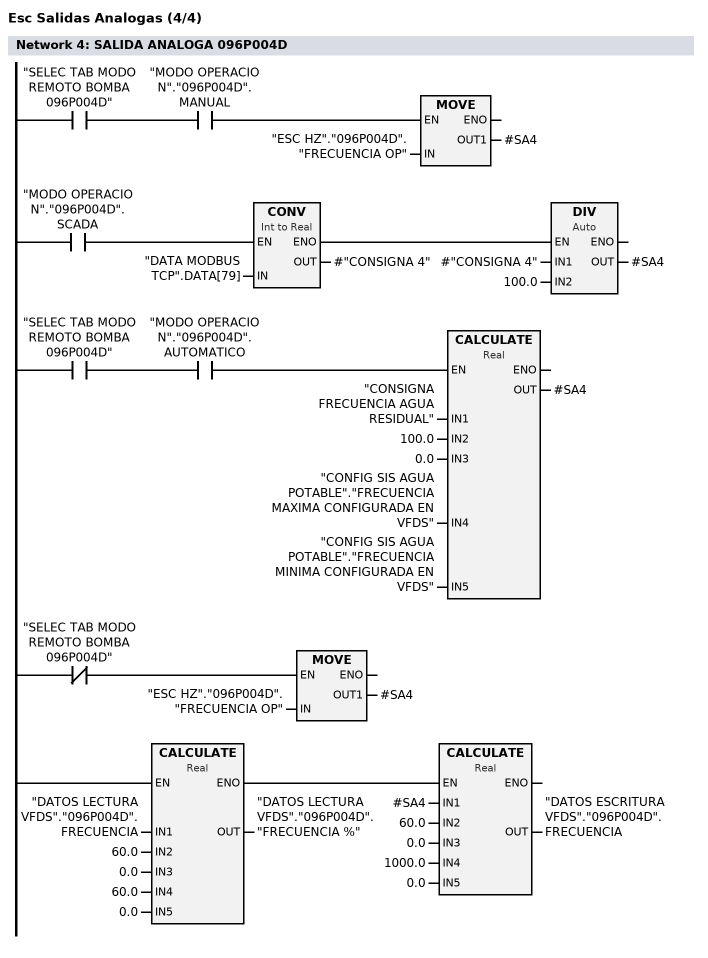
   RUNG wire#powerrail
      Contact( "SELEC TAB MODO REMOTO BOMBA 096P004D" )
      Contact( "MODO OPERACION"."096P004D".MANUAL )
      Move(in := "ESC HZ"."096P004D"."FRECUENCIA OP", out1 => #SA4)
   END_RUNG
   RUNG wire#powerrail
      Contact( "MODO OPERACION"."096P004D".SCADA )
      { S7_Templates := "[SrcType := Int, DestType := Real]" } Convert(in := "DATA MODBUS TCP".DATA[79], out => #"CONSIGNA 4")
      Div(in1 := #"CONSIGNA 4", in2 := 100.0, out => #SA4)
   END_RUNG
   RUNG wire#powerrail
      Contact( "SELEC TAB MODO REMOTO BOMBA 096P004D" )
      Contact( "MODO OPERACION"."096P004D".AUTOMATICO )
      { S7_Templates := "SrcType := Real"; S7_Expression := "(((IN4-IN5)/(IN2-IN3))*IN1)+(IN5-(((IN4-IN5)/(IN2-IN3))*IN3))" } Calculate(in1 := "CONSIGNA FRECUENCIA AGUA RESIDUAL", in2 := 100.0, in3 := 0.0, in4 := "CONFIG SIS AGUA POTABLE"."FRECUENCIA MAXIMA CONFIGURADA EN VFDS", in5 := "CONFIG SIS AGUA POTABLE"."FRECUENCIA MINIMA CONFIGURADA EN VFDS", out => #SA4)
   END_RUNG
   RUNG wire#powerrail
      I_Contact( "SELEC TAB MODO REMOTO BOMBA 096P004D" )
      Move(in := "ESC HZ"."096P004D"."FRECUENCIA OP", out1 => #SA4)
   END_RUNG
   RUNG wire#powerrail
      { S7_Templates := "SrcType := Real"; S7_Expression := "(((IN4-IN5)/(IN2-IN3))*IN1)+(IN5-(((IN4-IN5)/(IN2-IN3))*IN3))" } Calculate(in1 := "DATOS LECTURA VFDS"."096P004D".FRECUENCIA, in2 := 60.0, in3 := 0.0, in4 := 60.0, in5 := 0.0, out => "DATOS LECTURA VFDS"."096P004D"."FRECUENCIA %")
      { S7_Templates := "SrcType := Real"; S7_Expression := "(((IN4-IN5)/(IN2-IN3))*IN1)+(IN5-(((IN4-IN5)/(IN2-IN3))*IN3))" } Calculate(in1 := #SA4, in2 := 60.0, in3 := 0.0, in4 := 1000.0, in5 := 0.0, out => "DATOS ESCRITURA VFDS"."096P004D".FRECUENCIA)
   END_RUNG
   // the same network as SCL:
   IF "SELEC TAB MODO REMOTO BOMBA 096P004D" AND "MODO OPERACION"."096P004D".MANUAL THEN
       #SA4 := "ESC HZ"."096P004D"."FRECUENCIA OP";
   END_IF;
   IF "MODO OPERACION"."096P004D".SCADA THEN
       #"CONSIGNA 4" := INT_TO_REAL("DATA MODBUS TCP".DATA[79]);
       #SA4 := #"CONSIGNA 4" / 100.0;
   END_IF;
   IF "SELEC TAB MODO REMOTO BOMBA 096P004D" AND "MODO OPERACION"."096P004D".AUTOMATICO THEN
       #SA4 := ((("CONFIG SIS AGUA POTABLE"."FRECUENCIA MAXIMA CONFIGURADA EN VFDS"-"CONFIG SIS AGUA POTABLE"."FRECUENCIA MINIMA CONFIGURADA EN VFDS")/(100.0-0.0))*"CONSIGNA FRECUENCIA AGUA RESIDUAL")+("CONFIG SIS AGUA POTABLE"."FRECUENCIA MINIMA CONFIGURADA EN VFDS"-((("CONFIG SIS AGUA POTABLE"."FRECUENCIA MAXIMA CONFIGURADA EN VFDS"-"CONFIG SIS AGUA POTABLE"."FRECUENCIA MINIMA CONFIGURADA EN VFDS")/(100.0-0.0))*0.0));
   END_IF;
   IF NOT "SELEC TAB MODO REMOTO BOMBA 096P004D" THEN #SA4 := "ESC HZ"."096P004D"."FRECUENCIA OP"; END_IF;
   "DATOS LECTURA VFDS"."096P004D"."FRECUENCIA %" := (((60.0-0.0)/(60.0-0.0))*"DATOS LECTURA VFDS"."096P004D".FRECUENCIA)+(0.0-(((60.0-0.0)/(60.0-0.0))*0.0));
   "DATOS ESCRITURA VFDS"."096P004D".FRECUENCIA := (((1000.0-0.0)/(60.0-0.0))*#SA4)+(0.0-(((1000.0-0.0)/(60.0-0.0))*0.0));
END_REGION
END_FUNCTION

ORGANIZATION_BLOCK "Main"   // OB1, LAD, ProgramCycle
TITLE = "Main Program Sweep (Cycle)"
{ S7_Optimized_Access := 'TRUE' }
VERSION : 0.1
   VAR_INPUT
      Initial_Call : Bool;   // Initial call of this OB
      Remanence : Bool;   // =True, if remanent data are available
   END_VAR
   VAR_TEMP   // added for the SCL form of the ladder/FBD networks
      _w1 : Bool;
      _w2 : Bool;
   END_VAR
BEGIN

REGION Network 1
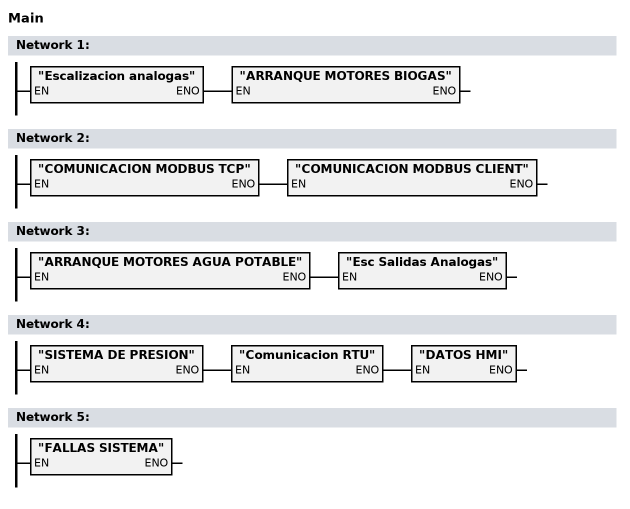
   RUNG wire#powerrail
      "Escalizacion analogas"()
      "ARRANQUE MOTORES BIOGAS"()
   END_RUNG
   // the same network as SCL:
   "Escalizacion analogas"(ENO => #_w1);
   IF #_w1 THEN "ARRANQUE MOTORES BIOGAS"(); END_IF;
END_REGION

REGION Network 2
   RUNG wire#powerrail
      "COMUNICACION MODBUS TCP"()
      "COMUNICACION MODBUS CLIENT"()
   END_RUNG
   // the same network as SCL:
   "COMUNICACION MODBUS TCP"(ENO => #_w1);
   IF #_w1 THEN "COMUNICACION MODBUS CLIENT"(); END_IF;
END_REGION

REGION Network 3
   RUNG wire#powerrail
      "ARRANQUE MOTORES AGUA POTABLE"()
      "Esc Salidas Analogas"()
   END_RUNG
   // the same network as SCL:
   "ARRANQUE MOTORES AGUA POTABLE"(ENO => #_w1);
   IF #_w1 THEN "Esc Salidas Analogas"(); END_IF;
END_REGION

REGION Network 4
   RUNG wire#powerrail
      "SISTEMA DE PRESION"()
      "Comunicacion RTU"()
      "DATOS HMI"()
   END_RUNG
   // the same network as SCL:
   "SISTEMA DE PRESION"(ENO => #_w1);
   "Comunicacion RTU"(EN := #_w1, ENO => #_w2);
   IF #_w2 THEN "DATOS HMI"(); END_IF;
END_REGION

REGION Network 5
   RUNG wire#powerrail
      "FALLAS SISTEMA"()
   END_RUNG
   // the same network as SCL:
   "FALLAS SISTEMA"();
END_REGION
END_ORGANIZATION_BLOCK

ORGANIZATION_BLOCK "PIDS"   // OB30, LAD, CyclicInterrupt
{ S7_Optimized_Access := 'TRUE' }
VERSION : 0.1
   VAR_INPUT
      Initial_Call : Bool;   // Initial call of this OB
      Event_Count : Int;   // Events discarded
   END_VAR
   VAR_TEMP
      SETPOINT : Real;
      SETPOINT2 : Real;
   END_VAR
BEGIN

REGION Network 1
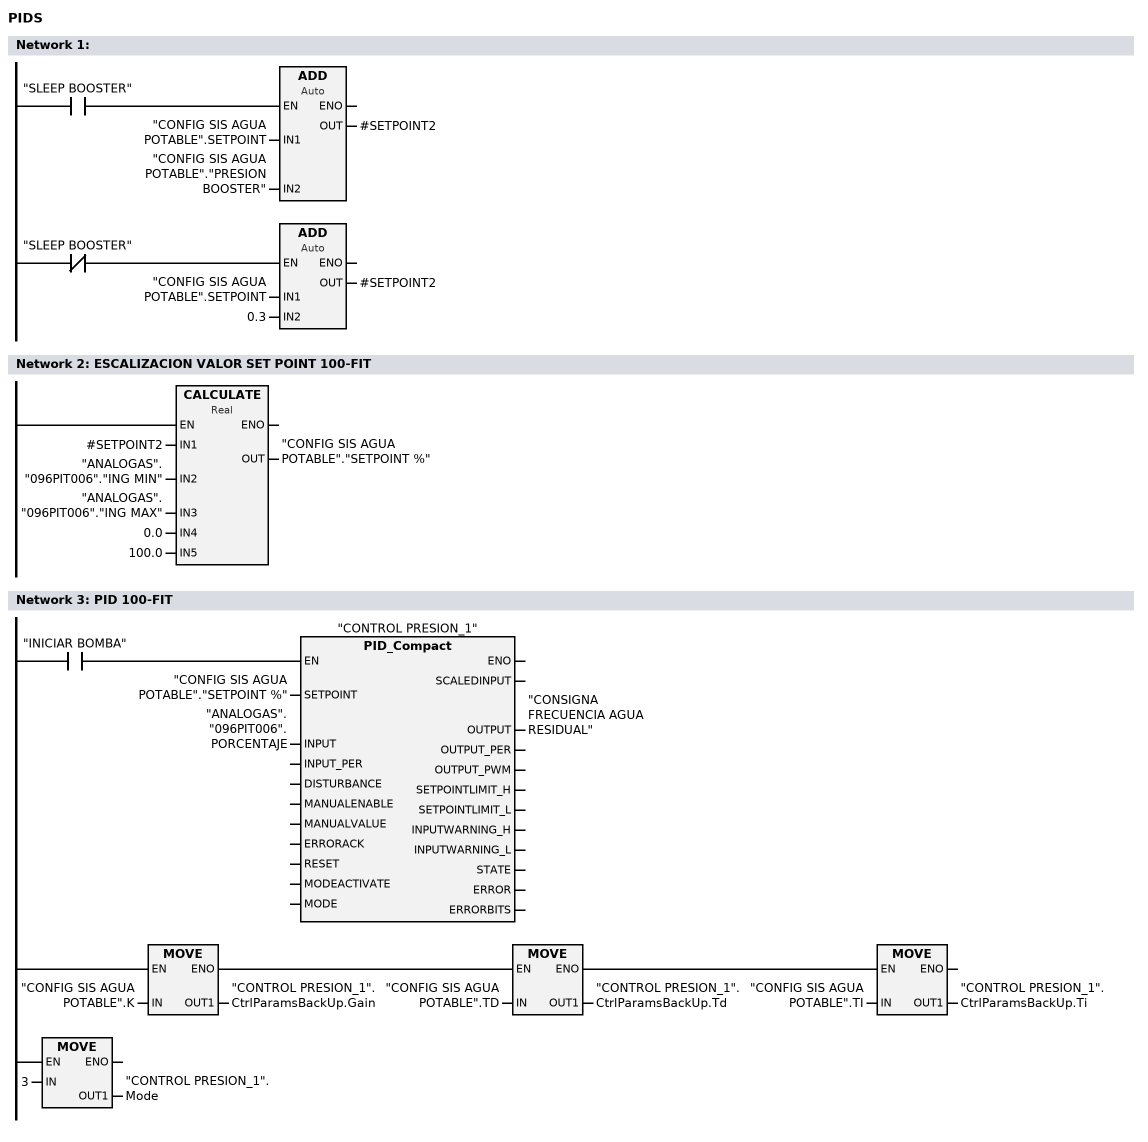
   RUNG wire#powerrail
      Contact( "SLEEP BOOSTER" )
      Add(in1 := "CONFIG SIS AGUA POTABLE".SETPOINT, in2 := "CONFIG SIS AGUA POTABLE"."PRESION BOOSTER", out => #SETPOINT2)
   END_RUNG
   RUNG wire#powerrail
      I_Contact( "SLEEP BOOSTER" )
      Add(in1 := "CONFIG SIS AGUA POTABLE".SETPOINT, in2 := 0.3, out => #SETPOINT2)
   END_RUNG
   // the same network as SCL:
   IF "SLEEP BOOSTER" THEN
       #SETPOINT2 := "CONFIG SIS AGUA POTABLE".SETPOINT + "CONFIG SIS AGUA POTABLE"."PRESION BOOSTER";
   END_IF;
   IF NOT "SLEEP BOOSTER" THEN #SETPOINT2 := "CONFIG SIS AGUA POTABLE".SETPOINT + 0.3; END_IF;
END_REGION

REGION Network 2: ESCALIZACION VALOR SET POINT 100-FIT
   RUNG wire#powerrail
      { S7_Templates := "SrcType := Real"; S7_Expression := "(((IN5-IN4)/(IN3-IN2))*IN1)+(IN4-((IN5-IN4)/(IN3-IN2)*IN2))" } Calculate(in1 := #SETPOINT2, in2 := "ANALOGAS"."096PIT006"."ING MIN", in3 := "ANALOGAS"."096PIT006"."ING MAX", in4 := 0.0, in5 := 100.0, out => "CONFIG SIS AGUA POTABLE"."SETPOINT %")
   END_RUNG
   // the same network as SCL:
   "CONFIG SIS AGUA POTABLE"."SETPOINT %" := (((100.0-0.0)/("ANALOGAS"."096PIT006"."ING MAX"-"ANALOGAS"."096PIT006"."ING MIN"))*#SETPOINT2)+(0.0-((100.0-0.0)/("ANALOGAS"."096PIT006"."ING MAX"-"ANALOGAS"."096PIT006"."ING MIN")*"ANALOGAS"."096PIT006"."ING MIN"));
END_REGION

REGION Network 3: PID 100-FIT
   IF "INICIAR BOMBA" THEN
       "CONTROL PRESION_1"(Setpoint := "CONFIG SIS AGUA POTABLE"."SETPOINT %",   // PID_Compact
                           Input := "ANALOGAS"."096PIT006".PORCENTAJE,
                           Output => "CONSIGNA FRECUENCIA AGUA RESIDUAL");
   END_IF;
   "CONTROL PRESION_1".CtrlParamsBackUp.Gain := "CONFIG SIS AGUA POTABLE".K;
   "CONTROL PRESION_1".CtrlParamsBackUp.Td := "CONFIG SIS AGUA POTABLE".TD;
   "CONTROL PRESION_1".CtrlParamsBackUp.Ti := "CONFIG SIS AGUA POTABLE".TI;
   "CONTROL PRESION_1".Mode := 3;
END_REGION
END_ORGANIZATION_BLOCK